TYPE checkInputVariable :
STRUCT
	EmergencyStop:BOOL;
	m_cartDriverInput :ARRAY[1..g_cartJntNum] OF ST_MotorInputs; 
	m_cartDriverOutput :ARRAY[1..g_cartJntNum] OF ST_MotorOutputs;
	m_slaveDriverInput :ARRAY[1..g_sJntNum] OF ST_MotorInputs; 
	m_slaveDriverOutput :ARRAY[1..g_sJntNum] OF ST_MotorOutputs;
	m_setupDriverInput :ARRAY[1..g_setupJntNum] OF ST_MotorInputs; 
	m_setupDriverOutput :ARRAY[1..g_setupJntNum] OF ST_MotorOutputs;
	
	m_EtherCATState:ARRAY [1..g_maxArmJoint] OF ST_EtherCATState;		
	m_rcpCheck : BOOL;
	m_spacePoseErr : vec6d;				
	m_cmdArmPos : 	vec6d;		
	m_instruOpenAngle:LREAL;		
	
	m_promptStatus:ARRAY [1..30] OF BOOL;
	m_promptLocation:ARRAY [1..30] OF UDINT;
	
	
	SlaveStopButton:BOOL;
	PCStopButton :UINT;
	MasterStopButton :BOOL;
	
	m_cartEtherCATState:ARRAY [1..g_maxCartJoint] OF ST_EtherCATState;
END_STRUCT
END_TYPE

(* stored: Version 1.1.0.1, ProductVersion 3.1.4024.11
   DUT checkInputVariable: Id {f641bcc5-1597-4d0c-903e-ba4da9cf7cc3} *)
